FUNCTION_BLOCK TurnTable
VAR_INPUT

	TT_0_Deg  			: BOOL;						//TurnTable at 0 degree
	TT_180_Deg 			: BOOL;						//TurnTable at 180 degree
	Part_Load_Comp 		: BOOL;						//OP710 Part Load Complete
	Part_Unload_Comp 	: BOOL;						//OP710 Part Unload Complete
	Pickup_Comp 		: BOOL;						//Robot Part Pickup Complete
	Roller_Down			: BOOL;						//Roller door Down position
	Roller_Up			: BOOL;						//Roller door Up position
	Fix_Home_Position 	: BOOL;
	Fix_Work_Position 	: BOOL;
	TR_0_Deg  			: BOOL;						//Trunnion at 0 degree
END_VAR

VAR_OUTPUT
	TT_0_Deg_Cmd  : BOOL;						//Trunnion rotate to 0 degree
	TT_180_Deg_Cmd : BOOL;						//Trunnion rotate to 180 degree
END_VAR

VAR
	TT_Rot_Delay : ARRAY [0..5] OF TON;							// TurnTable rotation delay
END_VAR

CASE Fix_Sel OF
	
	0: 

IF (TT_0_Deg AND TR_0_Deg AND Part_Load_Comp AND Fix_Work_Position AND Roller_Down AND Start_Pb) THEN
	TT_180_Deg_Cmd := TRUE;
	TT_Rot_Delay[0](IN:= TT_180_Deg_Cmd , PT:= T#1S, Q=> , ET=> );
	IF TT_Rot_Delay[0].Q THEN
	TT_0_Deg := FALSE;
	TT_180_Deg := TRUE;
	TT_180_Deg_Cmd := FALSE;
	END_IF	
ELSIF (TT_180_Deg AND Pickup_Comp AND Roller_Up AND Fix_Home_Position) THEN
	TT_0_Deg_Cmd := TRUE;
	TT_Rot_Delay[1](IN:= TT_0_Deg_Cmd , PT:= T#1S, Q=> , ET=> );
	IF TT_Rot_Delay[1].Q THEN
	TT_180_Deg := FALSE;
	TT_0_Deg := TRUE;
	TT_0_Deg_Cmd := FALSE;
	END_IF
END_IF
	Fix_Sel := 0;

	1: 

IF (TT_180_Deg AND TR_0_Deg AND Part_Load_Comp AND Fix_Work_Position AND Roller_Down AND Start_Pb) THEN
	TT_180_Deg_Cmd := TRUE;
	TT_Rot_Delay[2](IN:= TT_180_Deg_Cmd , PT:= T#1S, Q=> , ET=> );
	IF TT_Rot_Delay[2].Q THEN
	TT_0_Deg := FALSE;
	TT_180_Deg := TRUE;
	TT_180_Deg_Cmd := FALSE;
	END_IF	
ELSIF (TT_0_Deg AND Pickup_Comp AND Roller_Up AND Fix_Home_Position) THEN
	TT_180_Deg_Cmd := TRUE;
	TT_Rot_Delay[3](IN:= TT_180_Deg_Cmd , PT:= T#1S, Q=> , ET=> );
	IF TT_Rot_Delay[3].Q THEN
	TT_0_Deg := FALSE;
	TT_180_Deg := TRUE;
	TT_180_Deg_Cmd := FALSE;
	END_IF
END_IF
	Fix_Sel := 1;

END_CASE

END_FUNCTION_BLOCK

(* stored: Version 1.1.0.1, ProductVersion 3.1.4024.16
   POU TurnTable: Id {e1709711-f1ac-4ca3-b4f6-ce31c81ac309}, SpecialFunc None *)
